FUNCTION AllElementsEqualTo : BOOL
VAR_IN_OUT
	arr : ARRAY[*] OF INT;
END_VAR
VAR_INPUT
	firstIndex : SINT;
	lastIndex : SINT;
	value : INT;
END_VAR
VAR
	i : SINT := 0;
END_VAR

FOR i:=firstIndex TO lastIndex BY 1 DO
	IF NOT arr[i] = value THEN
		allElementsEqualTo := FALSE;
		RETURN;
	END_IF
END_FOR

allElementsEqualTo := TRUE;
RETURN;

END_FUNCTION

(* stored: Version 1.1.0.1, ProductVersion 3.1.4024.11
   POU AllElementsEqualTo: Id {26fdef38-f4a7-4280-ad00-fa6835f22b30}, SpecialFunc None *)
